(* CODESYS project CodexDashboard.export

Project tree, tasks and I/O mapping:
  visualisation CodexDashboard
*)

// /CodexDashboard
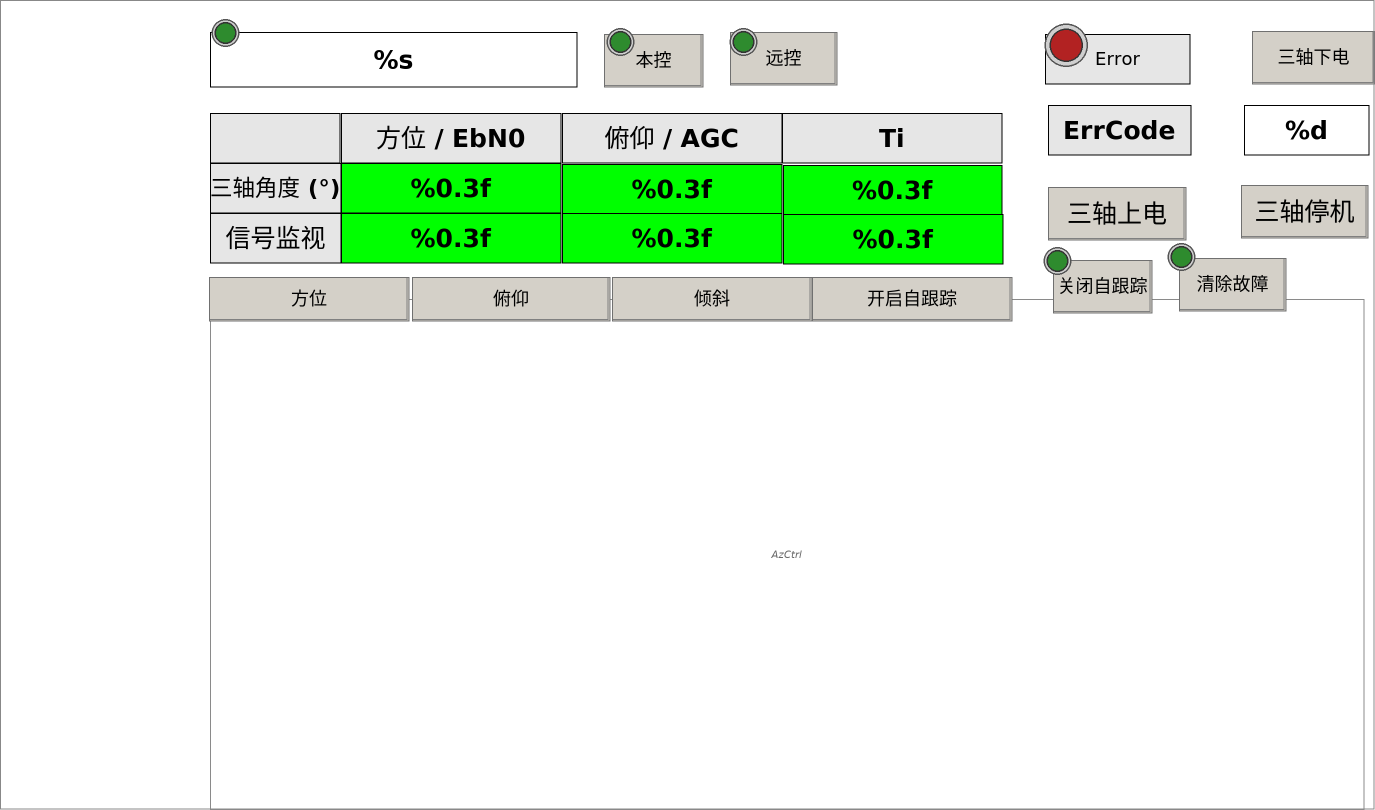
VISUALIZATION CodexDashboard  // 1375x810
    Rectangle (210,32 367x55), "%s", text variable: RealTimePosCal.dtReal
    Button (604,34 99x53), "本控"
        OnMouseClick: execute { GVL.bLocalCtrl:=TRUE; }
    Button (730,32 107x53), "远控"
        OnMouseClick: execute { GVL.bLocalCtrl:=FALSE; }
    Lamp1 (596,26 49x32), variable: GVL.bLocalCtrl, style: Lamp-Lamp1-Green
    Lamp1 (721,26 45x32), variable: NOT(GVL.bLocalCtrl), style: Lamp-Lamp1-Green
    Rectangle (341,113 220x50), "方位 / EbN0"
    Rectangle (562,113 220x50), "俯仰 / AGC"
    Rectangle (210,163 131x50), "三轴角度 (°)"
    Rectangle (341,163 220x50), "%0.3f", text variable: GVL.rFctPosReal_2*(-1)
    Rectangle (562,164 220x50), "%0.3f", text variable: GVL.rFctPosReal_1-90
    Rectangle (210,113 130x50)
    Rectangle (210,213 131x50), "信号监视"
    Rectangle (341,213 220x50), "%0.3f", text variable: READ_485.Chan1EB_N0
    Rectangle (562,213 220x50), "%0.3f", text variable: GVL.Chan1AGC
    Lamp1 (203,17 45x32), variable: TimeCase.Triger, style: Lamp-Lamp1-Green
    Rectangle (1045,34 145x50), "Error"
    Lamp1 (1026,20 80x50), variable: Az_ctrl_1.bVisError, style: Lamp-Lamp1-Red
    Button (1048,187 138x53), "三轴上电"
        OnMouseClick: execute {
            GVL.bLocalCtrl:=TRUE;
            GVL.Axis1Local.iMode:=1;
            GVL.Axis2Local.iMode:=1;
            GVL.Axis3Local.iMode:=1;
        }
    Button (1241,185 127x53), "三轴停机"
        OnMouseClick: execute {
            GVL.bLocalCtrl:=TRUE;
            GVL.Axis1Local.iMode:=7;
            GVL.Axis2Local.iMode:=7;
            GVL.Axis3Local.iMode:=7;
        }
    Rectangle (1048,105 143x50), "ErrCode"
    Rectangle (1244,105 125x50), "%d", text variable: GVL.Error_code
    Button (1252,31 123x53), "三轴下电"
        OnMouseClick: execute {
            GVL.bLocalCtrl:=TRUE;
            GVL.bStartLocalAutoTrack:=FALSE;
            GVL.Axis1Local.iMode:=0;
            GVL.Axis2Local.iMode:=0;
            GVL.Axis3Local.iMode:=0;
        }
    Rectangle (782,113 220x50), "Ti"
    Rectangle (783,165 219x50), "%0.3f", text variable: GVL.rFctPosReal_3*(-1)
    Rectangle (783,214 220x50), "%0.3f", text variable: GVL.rFctVelReal_3*(-1)
    TabControl (210,299 1154x511), frame switch variable: GVL.iVisualSwitch
        shows AzCtrl()
        shows ElCtrl()
        shows TlCtrl()
        shows north()
        shows IOtest()
        shows IOState()
    Button (209,277 200x44), "方位", input disabled if: GVL.bAzVisable
        OnMouseClick: execute {
            GVL.bAzVisable:=TRUE;
            GVL.bElVisable:=FALSE;
            GVL.bTlVisable:=FALSE;
            GVL.bLocalAutoTrackVis:=FALSE;
            GVL.iVisualSwitch:=0;
        }
    Button (412,277 198x44), "俯仰", input disabled if: GVL.bElVisable
        OnMouseClick: execute {
            GVL.bAzVisable:=FALSE;
            GVL.bElVisable:=TRUE;
            GVL.bTlVisable:=FALSE;
            GVL.bLocalAutoTrackVis:=FALSE;
            GVL.iVisualSwitch:=1;
        }
    Button (612,277 200x44), "倾斜", input disabled if: GVL.bTlVisable
        OnMouseClick: execute {
            GVL.bAzVisable:=FALSE;
            GVL.bElVisable:=FALSE;
            GVL.bTlVisable:=TRUE;
            GVL.bLocalAutoTrackVis:=FALSE;
            GVL.iVisualSwitch:=2;
        }
    Button (812,277 200x44), "开启自跟踪", input disabled if: GVL.bLocalAutoTrackVis
        OnMouseClick: execute {
            GVL.bLocalCtrl:=TRUE;
            GVL.bStartLocalAutoTrack:=TRUE;
            GVL.Axis1Local.iMode:=4;
            GVL.Axis2Local.iMode:=4;
            GVL.Axis3Local.iMode:=4;
        }
    Button (1053,260 99x53), "关闭自跟踪"
        OnMouseClick: execute { GVL.bStartLocalAutoTrack:=FALSE; }
    Button (1179,258 107x53), "清除故障"
        OnMouseClick: execute { GVL.bError_Reset:=TRUE; }
    Lamp1 (1033,245 49x32), variable: NOT(GVL.bTimeSwich), style: Lamp-Lamp1-Green
    Lamp1 (1159,241 45x32), variable: GVL.bTimeSwich, style: Lamp-Lamp1-Green
END_VISUALIZATION
